{attribute 'qualified_only'}
{attribute 'strict'}
{attribute 'to_string'}
TYPE E_ControlMode :
(
	Manual := 0,
	Recipe := 1,
	Priority := 2
);
END_TYPE

(* stored: Version 1.1.0.1, ProductVersion 3.1.4026.11
   DUT E_ControlMode: Id {043536e2-aedf-4c82-8eab-ab0e4bdacad6} *)
